{attribute 'TcGenerated'}
{attribute 'no-analysis'}
{attribute 'linkalways'}
// This function has been automatically generated from the project information.
VAR_GLOBAL CONSTANT
	{attribute 'const_non_replaced'}
	stLibVersion_LCLSVacuumLib : ST_LibVersion := (iMajor := 1, iMinor := 12, iBuild := 6969, iRevision := 0, sVersion := '1.12.6969');
END_VAR

(* stored: Version 1.1.0.1, ProductVersion 3.1.4022.18
   GVL Global_Version: Id {d92ec28a-e0bd-46af-b967-3e6dee49e59a} *)
